(* IEC 61131-3 sources: learning-path/07_unit_testing/exercises/solutions/2_testing_classes_solution, 1 file *)

(* ---- test.st ---- *)
USING AxUnit.Assert;
USING Counter;

NAMESPACE Test
    {TestFixture}
    CLASS CounterTest
        VAR
            simpleCounter : SimpleCounter;
        END_VAR

        {Test}
        METHOD PUBLIC CountFrom2To4
            simpleCounter.SetCurrentValue(2);
            simpleCounter.CountUp();
            simpleCounter.CountUp();
            Equal(actual := simpleCounter.GetCurrentValue(), expected := 4);
        END_METHOD
    END_CLASS
END_NAMESPACE
